Staubli VAL3: refreshStatic.pgx

program refreshStatic()
  local string l_sMenu
  local num i
  local string l_sMessage
  local string l_sName
begin
  title("PE_Solar")
    l_sMenu="模拟,复位,,,,,,"
  // define the menu
  call use:stringToArray(l_sMenu,sMenu)
    // set the menu
  call use:setMenu(sMenu,true,2)
  call use:getMenu(sMenu,bButton)
end
